{attribute 'qualified_only'}
{attribute 'strict'}
TYPE E_DTType : 
(
	NotInitialized := 0,
	BOOL_,
	BYTE_,
	WORD_,
	DWORD_,
	SINT_,
	USINT_,
	INT_,
	UINT_,
	DINT_,
	UDINT_,
	LINT_,
	ULINT_,
	REAL_,
	LREAL_,
	LWORD_
) ;
END_TYPE

(* stored: DUT E_DTType: Id 9903e9d1-ad46-4106-8a38-e0fb8fc82196 *)
